// Parses a 64-bit little-endian integer.
FUNCTION F_ParseRawLittleEndian64 : HRESULT
VAR_INPUT
    stBuffer : ST_Span; 
END_VAR
VAR_IN_OUT
    stState : ST_ParserInternalState;
END_VAR
VAR_OUTPUT
    nValue : ULINT;
END_VAR
VAR CONSTANT
    cLength : UDINT := SIZEOF(nValue);
END_VAR


F_ParseRawLittleEndian64 := S_OK;

IF stState.nBufferSize - stState.nBufferPos < cLength THEN
    F_ParseRawLittleEndian64 := stState.eParserErrorCode := E_ParserErrorCode.TruncatedMessage;
    stState.bError := TRUE;
    RETURN;
END_IF

MEMCPY(destAddr:= ADR(nValue), srcAddr:=stBuffer.pBuffer + stState.nBufferPos, n:= cLength);
stState.nBufferPos := stState.nBufferPos + cLength;

END_FUNCTION

(* stored: Version 1.1.0.1
   POU F_ParseRawLittleEndian64: Id {be6bf815-3ecb-4adf-a4c6-a29e7ee5429d}, SpecialFunc None *)
